// TwinCAT 3 PLC project MAS418_PLC
// ProgramVersion: 3.1.4023.0
// libraries:
//   Tc2_Standard, * (Beckhoff Automation GmbH)
//   Tc2_System, * (Beckhoff Automation GmbH)
//   Tc3_Module, * (Beckhoff Automation GmbH)
//   VisuDialogs, * (System)
// project tree:
//   / GlobalTextList.TcGTLO, PlcTask.TcTTO, Visualization Manager.TcVMO (not stored)
//   POUs/ MAIN.TcPOU
//   VISUs/ Visualization.TcVIS
// real-time tasks:
//   TASK PlcTask: cycle T#10ms, priority 20, ADS port 350

CONFIGURATION MAS418_PLC
    RESOURCE PLC ON TwinCAT3
        TASK PlcTask(INTERVAL := T#10ms, PRIORITY := 20);
        PROGRAM MAIN WITH PlcTask : MAIN;
    END_RESOURCE
END_CONFIGURATION

// ---- POUs/MAIN.TcPOU
PROGRAM MAIN
VAR
	bEnable : BOOL;
	bStart : BOOL;
	nINT : INT := -32768;
	nUINT : UINT := 65535;
	fREAL : REAL := 255.255;
	sPowerStatus: STRING := 'Power Off';
	nFloatConversion : INT := 500;
	fFloatConversion : LREAL;
	nIntConversion : INT;
	fIntConversion : LREAL := 45.67;
	
END_VAR

bEnable := bStart;
fFloatConversion := INT_TO_LREAL(nFloatConversion);
nIntConversion := LREAL_TO_INT(fIntConversion);

END_PROGRAM

// ---- GlobalTextList.TcGTLO
TEXTLIST GlobalTextList
  444 = '%s'
  82 = 'BOOL'
  818 = 'DataTypeTesting'
  998 = 'INT'
  741 = 'INT%i'
  261 = 'Power ON'
  880 = 'REAL'
  989 = 'REAL%f'
  345 = 'REAL%i'
  414 = 'STRING'
  568 = 'STRING%s'
  581 = 'UINT'
  95 = 'UINT%i'
END_TEXTLIST

// ---- VISUs/Visualization.TcVIS
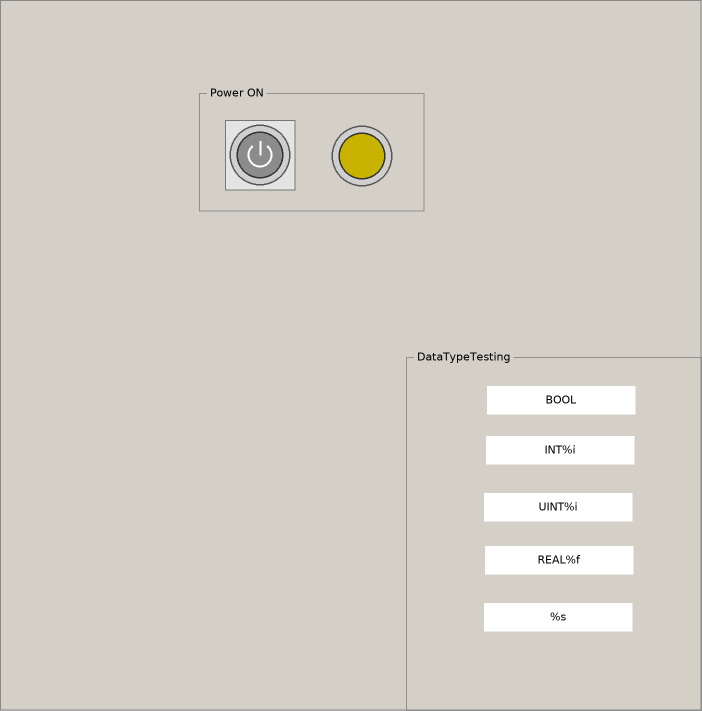
VISUALIZATION Visualization  // 702x711
    GroupBox (199,85 225x126), "Power ON"
        Lamp1 (128,36 70x70), variable: MAIN.bEnable, style: Lamp-Lamp1-Yellow
        PowerSwitch (26,35 70x70), variable: MAIN.bStart, behaviour: TOGGLE, style: Switch-PowerSwitch-Gray
    GroupBox (406,349 296x362), "DataTypeTesting"
        Textfield (80,36 150x30), "BOOL"
        Textfield (79,86 150x30), "INT%i", text variable: MAIN.nINT
        Textfield (77,143 150x30), "UINT%i", text variable: MAIN.nUINT
        Textfield (78,196 150x30), "REAL%f", text variable: MAIN.fREAL
            OnMouseDown: write the text variable via Default
        Textfield (77,253 150x30), "%s", text variable: MAIN.sPowerStatus
            OnMouseDown: write the text variable via Default
END_VISUALIZATION
